# EPICS substitutions: db/Beckhoff_7XXX/ecmcEL7041.substitutions
file "ecmcEL7031-chX.template"
{
  pattern {CH_ID}
          {01   }
}

file "ecmcEL5101-chX.template"
{
  pattern {CH_ID}
          {01   }
}
